// TwinCAT 3 PLC project PLC
// ProgramVersion: 3.1.4026.17
// libraries:
//   Tc2_Standard, * (Beckhoff Automation GmbH)
//   Tc2_System, * (Beckhoff Automation GmbH)
// project tree:
//   / MAIN.TcPOU, PlcTask.TcTTO
//   POUs/ I_Base.TcIO, I_Mover.TcIO, I_ParameterPosition.TcIO, I_ParameterPositionGetter.TcIO, Mover.TcPOU, ParameterSet.TcPOU, InterfaceTaskExample.TcPOU, PointerTaskExample.TcPOU
// real-time tasks:
//   TASK PlcTask: cycle T#10ms, priority 20, ADS port 350

CONFIGURATION PLC
    RESOURCE PLC ON TwinCAT3
        TASK PlcTask(INTERVAL := T#10ms, PRIORITY := 20);
        PROGRAM MAIN WITH PlcTask : MAIN;
    END_RESOURCE
END_CONFIGURATION

// ---- POUs/I_Base.TcIO
INTERFACE I_Base EXTENDS __SYSTEM.IQueryInterface

END_INTERFACE

// ---- POUs/I_Mover.TcIO
INTERFACE I_Mover EXTENDS I_Base

{attribute 'monitoring':='call'}
PROPERTY Parameters : I_ParameterPosition
GET
END_GET
SET
END_SET
END_PROPERTY

{attribute 'monitoring':='call'}
PROPERTY Status : I_ParameterPositionGetter
GET
END_GET
END_PROPERTY

END_INTERFACE

// ---- POUs/I_ParameterPosition.TcIO
INTERFACE I_ParameterPosition EXTENDS I_ParameterPositionGetter

{attribute 'monitoring' := 'call'}
PROPERTY Position : LREAL
SET
END_SET
END_PROPERTY

END_INTERFACE

// ---- POUs/I_ParameterPositionGetter.TcIO
INTERFACE I_ParameterPositionGetter EXTENDS I_Base

{attribute 'monitoring' := 'call'}
PROPERTY Position : LREAL
GET
END_GET
END_PROPERTY

END_INTERFACE

// ---- MAIN.TcPOU
PROGRAM MAIN
VAR
	testMover : Mover;
END_VAR

testMover.CyclicLogic();

END_PROGRAM

// ---- POUs/Mover.TcPOU
FUNCTION_BLOCK Mover IMPLEMENTS I_Mover
VAR
	{attribute 'hide'}
	_Parameters : ParameterSet;
	{attribute 'hide'}
	_Status		: ParameterSet;
	{attribute 'hide'}
	_PointerExample : BOOL;
	testTask	: InterfaceTaskExample(_Parameters, _Status);
	pointerTask : PointerTaskExample(THIS^);
END_VAR

METHOD CyclicLogic
VAR_INPUT
END_VAR
IF _PointerExample THEN
	pointerTask.CyclicLogic();
	RETURN;
END_IF

testTask.CyclicLogic();
END_METHOD

{attribute 'monitoring':='call'}
PROPERTY Parameters : I_ParameterPosition
GET
Parameters := _Parameters;
END_GET
SET
END_SET
END_PROPERTY

{attribute 'monitoring':='call'}
PROPERTY PointerExample : BOOL
GET
PointerExample := _PointerExample;
END_GET
SET
_PointerExample := PointerExample;
END_SET
END_PROPERTY

{attribute 'monitoring':='call'}
PROPERTY Status : I_ParameterPositionGetter
GET
Status := _Status;
END_GET
END_PROPERTY

END_FUNCTION_BLOCK

// ---- POUs/ParameterSet.TcPOU
FUNCTION_BLOCK ParameterSet IMPLEMENTS I_ParameterPosition
VAR
	{attribute 'hide'}
	_Position : LREAL;
END_VAR

PROPERTY Position : LREAL
GET
Position := _Position;
END_GET
SET
_Position := Position;
END_SET
END_PROPERTY

END_FUNCTION_BLOCK

// ---- POUs/InterfaceTaskExample.TcPOU
FUNCTION_BLOCK InterfaceTaskExample
VAR
	_parameter : I_ParameterPosition;
	_status	   : I_ParameterPosition;
END_VAR

METHOD CyclicLogic
VAR_INPUT
END_VAR
IF _parameter = 0 OR _status = 0 THEN
	RETURN;
END_IF
_status.Position := _parameter.Position;
END_METHOD

//FB_Init is always available implicitly and it is used primarily for initialization.
//The return value is not evaluated. For a specific influence, you can also declare the
//methods explicitly and provide additional code there with the standard initialization
//code. You can evaluate the return value.
METHOD FB_Init: BOOL
VAR_INPUT
    bInitRetains: BOOL; // TRUE: the retain variables are initialized (reset warm / reset cold)
    bInCopyCode: BOOL;  // TRUE: the instance will be copied to the copy code afterward (online change)   
	Parameter : I_ParameterPosition;
	Status : I_ParameterPosition;
END_VAR
_parameter := Parameter;
_Status := Status;
END_METHOD

END_FUNCTION_BLOCK

// ---- POUs/PointerTaskExample.TcPOU
FUNCTION_BLOCK PointerTaskExample
VAR
	_parameter : I_ParameterPosition;
	_status	   : POINTER TO ParameterSet;
END_VAR

METHOD CyclicLogic
VAR_INPUT
END_VAR
IF _parameter = 0 OR _status = 0 THEN
	RETURN;
END_IF
_status^.Position := _parameter.Position;
END_METHOD

//FB_Init is always available implicitly and it is used primarily for initialization.
//The return value is not evaluated. For a specific influence, you can also declare the
//methods explicitly and provide additional code there with the standard initialization
//code. You can evaluate the return value.
METHOD FB_Init: BOOL
VAR_INPUT
    bInitRetains: BOOL; // TRUE: the retain variables are initialized (reset warm / reset cold)
    bInCopyCode: BOOL;  // TRUE: the instance will be copied to the copy code afterward (online change)   
	Mover : I_Mover;
END_VAR
_parameter := Mover.Parameters;
__QUERYPOINTER(Mover.Status,_Status);
END_METHOD

END_FUNCTION_BLOCK
